// TIA Portal V19 export
TYPE "udt_ZoneSafetyInterface"
// stored: Access Published, IsFailsafeCompliant true
   STRUCT
      Door_NormalStop : Bool;
      Door_SafeStop : Bool;
      Door_Opened : Bool;
      Door_EntryEnable : Bool;
   END_STRUCT;
END_TYPE
